// TIA Portal V19 export
TYPE "C406_STU_IF_CAD_TYPIC"
   STRUCT
      CMD_TOE { ExternalAccessible := 'False'; ExternalVisible := 'False'; ExternalWritable := 'False'} : Bool;   // Aansturing calamiteitendoorsteek Dicht
      CMD_OPEN { ExternalAccessible := 'False'; ExternalVisible := 'False'; ExternalWritable := 'False'} : Bool;   // Aansturing calamiteitendoorsteek Open
      CMD_RES { ExternalAccessible := 'False'; ExternalVisible := 'False'; ExternalWritable := 'False'} : Bool;   // Reset van de latched storingen
      CMD_SNS_RES { ExternalAccessible := 'False'; ExternalVisible := 'False'; ExternalWritable := 'False'} : Bool;   // Reset van de noodstop storingen
   END_STRUCT;
END_TYPE
